FUNCTION_BLOCK FB_HMI_LAKESHORE EXTENDS FB_HMI_COMPONENT
VAR_INPUT
    bConnected : BOOL;
END_VAR
VAR_OUTPUT
END_VAR
VAR_IN_OUT
    fbInstance : FB_METIS_LAKESHORE_336_TCP;
END_VAR
VAR
END_VAR

fbHealthStatus(
    bIsEnabled := bConnected,
    bIsGood := fbInstance.stat.nSubstate = E_RS_BASE_SUBSTATE.OP_MONITORING,
    bHasWarning := fbInstance.stat.bLocal);
                     
fbBusyStatus(
    bIsEnabled := bConnected,
    bIsBusy := fbInstance.stat.nSubstate = E_RS_BASE_SUBSTATE.NOTOP_INITIALIZING);

M_UpdateStatusColor();

END_FUNCTION_BLOCK

(* stored: Version 1.1.0.1, ProductVersion 3.1.4024.14
   POU FB_HMI_LAKESHORE: Id {e25329ba-1e78-40af-a51d-0181e9790c3a}, SpecialFunc None *)
